// Mitsubishi GX Works2 project: biomass   PLC: FX3U/FX3UC

PROGRAM MAIN
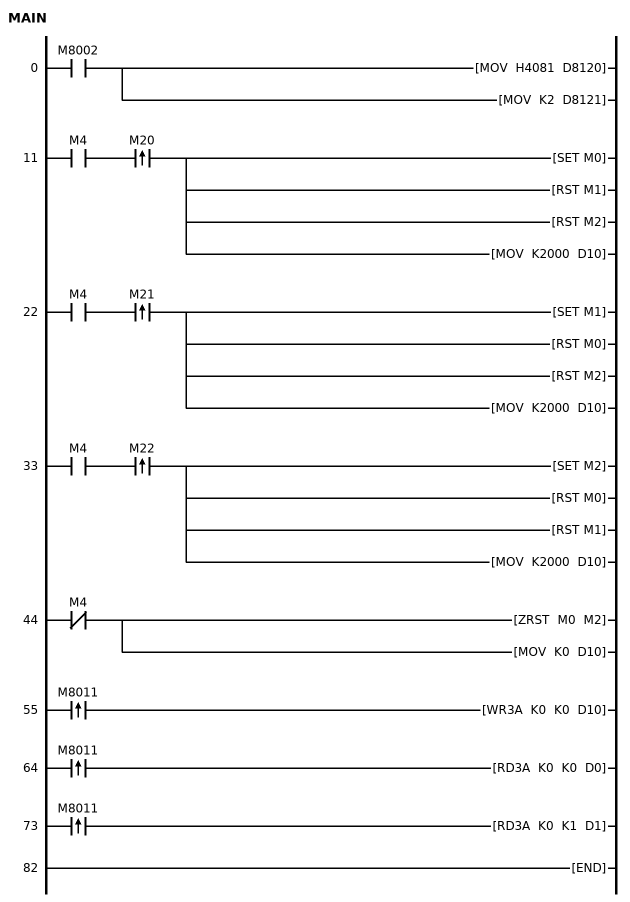
0     LD      M8002
      MOV     H4081 D8120
      MOV     K2 D8121
11    LD      M4
      ANDP    M20
      SET     M0
      RST     M1
      RST     M2
      MOV     K2000 D10
22    LD      M4
      ANDP    M21
      SET     M1
      RST     M0
      RST     M2
      MOV     K2000 D10
33    LD      M4
      ANDP    M22
      SET     M2
      RST     M0
      RST     M1
      MOV     K2000 D10
44    LDI     M4
      ZRST    M0 M2
      MOV     K0 D10
55    LDP     M8011
      WR3A    K0 K0 D10
64    LDP     M8011
      RD3A    K0 K0 D0
73    LDP     M8011
      RD3A    K0 K1 D1
82    END
END_PROGRAM
